Staubli VAL3: isEnable.pgx

public program isEnable(bool& x_bEnable[], string x_sItem)
  local num l_nSize
begin
  // check if is active
  x_bEnable=saveInOut:dInput[x_sItem].bEnable
end
